(* Logix 5000 project; controller STAT 1756-L72 rev 20.12; software revision 20.04; part 15 of 34 *)
(* tags used below, declared in another part *)
   AUX_P1P2 : BOOL;
   B10 : DINT[20];
   B14 : DINT[30];
   B15 : DINT[30];
   B16 : DINT[30];
   B17 : DINT[30];
   B3 : DINT[256];
   B9 : DINT[40];
   DateTime : DINT[7];   // DINT array tag for retrieve wallclock time through GSV created during conversion
   F8 : REAL[256];
   GEN_FOUT : BOOL;
   I1_005_Bit14 : ALIAS FOR I1[5].14;
   I1_005_Bit15 : ALIAS FOR I1[5].15;
   I1_008_Bit01 : ALIAS FOR I1[8].1;   // Hand Automaat stormbekken
   I1_009_Bit04 : ALIAS FOR I1[9].4;   // Pomp 1 in lijn
   I1_009_Bit08 : ALIAS FOR I1[9].8;   // Pomp 2 in lijn
   I1_009_Bit12 : ALIAS FOR I1[9].12;   // Pomp 3 in lijn
   I1_010_Bit05 : ALIAS FOR I1[10].5;   // Vlotterschak lal stormbekken
   I2_001_Bit07 : ALIAS FOR I2[1].7;   // Motor p11 lijn1 in dienst
   I2_001_Bit09 : ALIAS FOR I2[1].9;   // Motor p12 lijn1 in dienst
   I2_001_Bit11 : ALIAS FOR I2[1].11;   // Motor p13 lijn2 in dienst
   I2_001_Bit13 : ALIAS FOR I2[1].13;   // Motor p14 lijn2 in dienst
   I2_001_Bit15 : ALIAS FOR I2[1].15;   // Motor p15 lijn3 in dienst
   I3_000_Bit00 : ALIAS FOR I3[0].0;   // Motor p15 lijn3 thermische storing
   I3_000_Bit03 : ALIAS FOR I3[0].3;   // Motor p17 lijn4 in dienst
   I3_000_Bit05 : ALIAS FOR I3[0].5;   // Motor p18 lijn4 in dienst
   I3_000_Bit09 : ALIAS FOR I3[0].9;   // Motor pro 1 voedingpomp osmose 1 in driehoek
   I3_000_Bit13 : ALIAS FOR I3[0].13;   // Motor pro 2 voedingpomp osmose 2 in driehoek
   I3_001_Bit09 : ALIAS FOR I3[1].9;   // Motor voedingspomp osmose 3 in drie
   I4_000_Bit01 : ALIAS FOR I4[0].1;   // READY DRIVE P3
   I4_000_Bit04 : ALIAS FOR I4[0].4;   // Motor p4 in lijn in
   I4_000_Bit05 : ALIAS FOR I4[0].5;   // ready drive p4
   I5_001_Bit12 : ALIAS FOR I5[1].12;   // EV6_OPEN
   I5_001_Bit13 : ALIAS FOR I5[1].13;   // EV6_TOE
   I5_001_Bit14 : ALIAS FOR I5[1].14;   // EV7_TOE
   I5_001_Bit15 : ALIAS FOR I5[1].15;   // EV7_OPEN
   I6_000_Bit13 : ALIAS FOR I6[0].13;   // ES_EV2_IS_TOE
   I6_000_Bit14 : ALIAS FOR I6[0].14;   // ES_EV2_IS_OPEN
   I7_000_Bit07 : ALIAS FOR I7[0].7;   // hoog alarm ketel tampon
   I7_000_Bit08 : ALIAS FOR I7[0].8;   // midden alarm ketel tampon
   I7_000_Bit09 : ALIAS FOR I7[0].9;   // laag alarm ketel tampon
   I7_001_Bit08 : ALIAS FOR I7[1].8;   // q4 debietsmeting osmose 1 fout
   I8_000_Bit04 : ALIAS FOR I8[0].4;   // niveau kuip 20m hoog alarm
   I8_000_Bit06 : ALIAS FOR I8[0].6;   // niveau kuip 20m laag niv
   I9_000_Bit09 : ALIAS FOR I9[0].9;   // Hand_Auto CL7
   N11 : DINT[150];
   N12 : DINT[230];
   N13 : DINT[230];
   O15_001_Bit06 : ALIAS FOR O15[1].6;   // EV2 EV2
   O15_001_Bit07 : ALIAS FOR O15[1].7;   // EV3 EV3
   O15_001_Bit10 : ALIAS FOR O15[1].10;   // EV6 EV6
   O15_001_Bit11 : ALIAS FOR O15[1].11;   // EV7 EV7
   old_o13_3 : BOOL;
   T27 : TIMER[100];
   T4 : TIMER[200];
(* ibt, continued *)

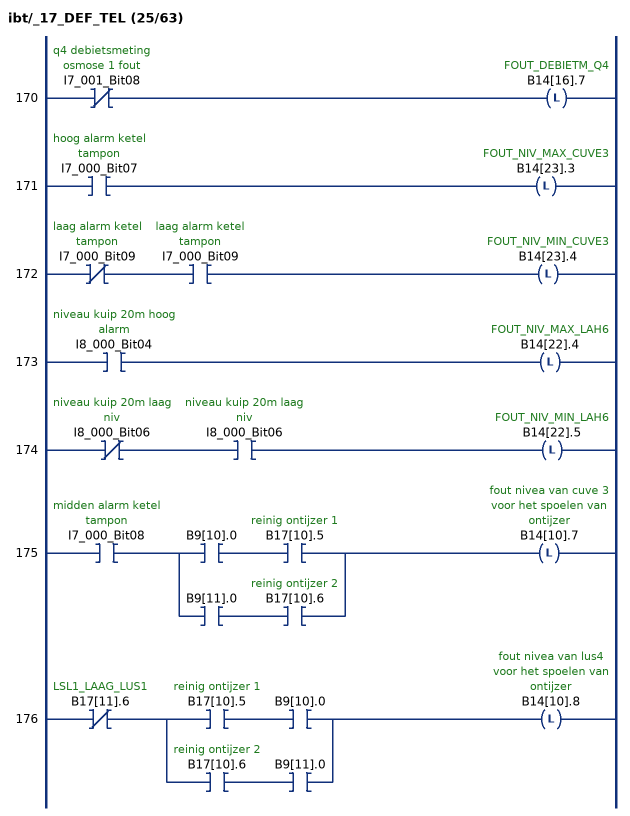
   [picture p249: ibt/_17_DEF_TEL rungs 170-176]
   170: XIO(I7_001_Bit08)OTL(B14[16].7);
   171: XIC(I7_000_Bit07)OTL(B14[23].3);
   172: XIO(I7_000_Bit09)XIC(I7_000_Bit09)OTL(B14[23].4);
   173: XIC(I8_000_Bit04)OTL(B14[22].4);
   174: XIO(I8_000_Bit06)XIC(I8_000_Bit06)OTL(B14[22].5);
   175: XIC(I7_000_Bit08)[XIC(B9[10].0) XIC(B17[10].5) ,XIC(B9[11].0) XIC(B17[10].6) ]OTL(B14[10].7);
   176: XIO(B17[11].6)[XIC(B17[10].5) XIC(B9[10].0) ,XIC(B17[10].6) XIC(B9[11].0) ]OTL(B14[10].8);
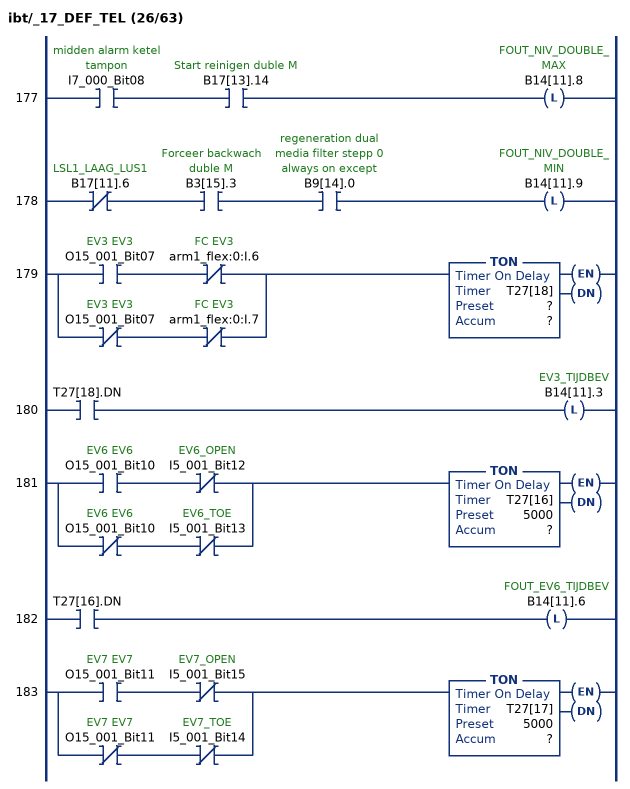
   177: XIC(I7_000_Bit08)XIC(B17[13].14)OTL(B14[11].8);
   178: XIO(B17[11].6)XIC(B3[15].3)XIC(B9[14].0)OTL(B14[11].9);
   179: [XIC(O15_001_Bit07) XIO(arm1_flex:0:I.6) ,XIO(O15_001_Bit07) XIO(arm1_flex:0:I.7) ]TON(T27[18],?,?);
   180: XIC(T27[18].DN)OTL(B14[11].3);
   181: [XIC(O15_001_Bit10) XIO(I5_001_Bit12) ,XIO(O15_001_Bit10) XIO(I5_001_Bit13) ]TON(T27[16],?,?);
   182: XIC(T27[16].DN)OTL(B14[11].6);
   183: [XIC(O15_001_Bit11) XIO(I5_001_Bit15) ,XIO(O15_001_Bit11) XIO(I5_001_Bit14) ]TON(T27[17],?,?);
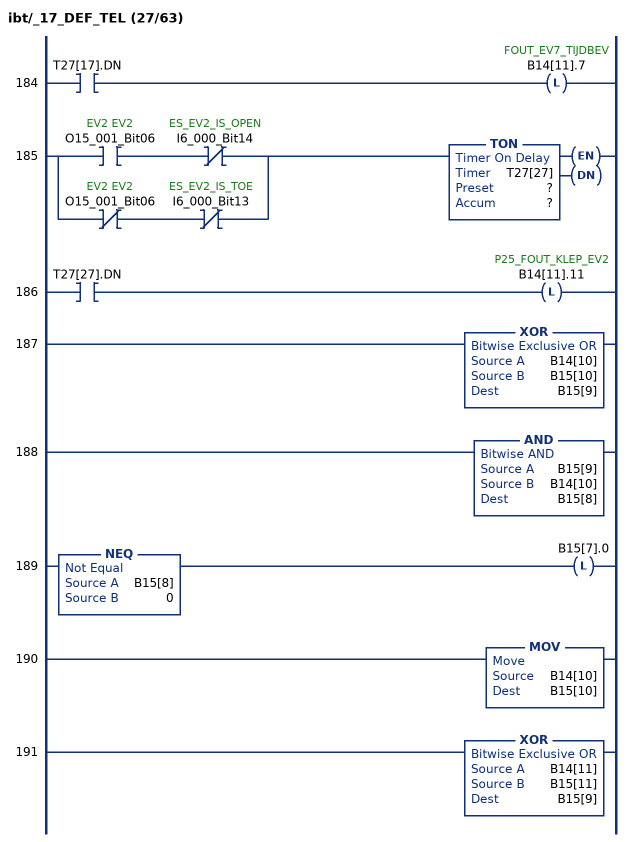
   184: XIC(T27[17].DN)OTL(B14[11].7);
   185: [XIC(O15_001_Bit06) XIO(I6_000_Bit14) ,XIO(O15_001_Bit06) XIO(I6_000_Bit13) ]TON(T27[27],?,?);
   186: XIC(T27[27].DN)OTL(B14[11].11);
   187: XOR(B14[10],B15[10],B15[9]);
   188: AND(B15[9],B14[10],B15[8]);
   189: NEQ(B15[8],0)OTL(B15[7].0);
   190: MOV(B14[10],B15[10]);
   191: XOR(B14[11],B15[11],B15[9]);
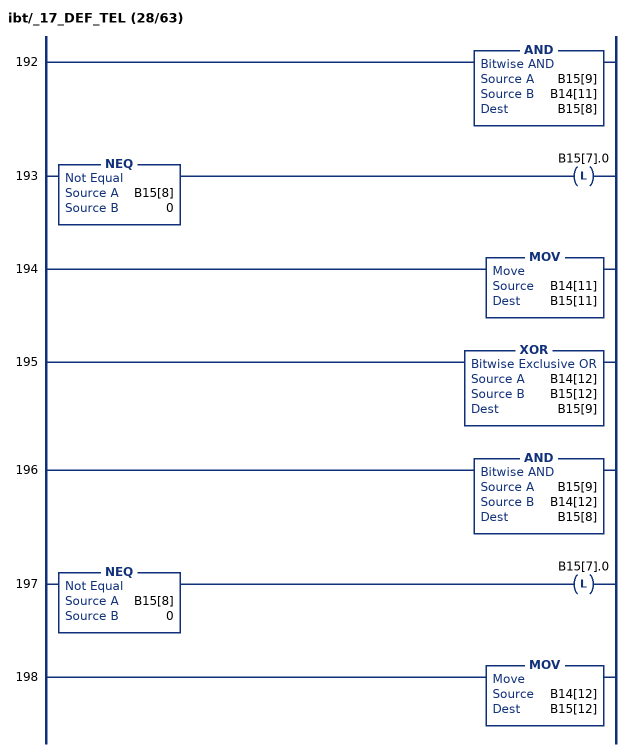
   192: AND(B15[9],B14[11],B15[8]);
   193: NEQ(B15[8],0)OTL(B15[7].0);
   194: MOV(B14[11],B15[11]);
   195: XOR(B14[12],B15[12],B15[9]);
   196: AND(B15[9],B14[12],B15[8]);
   197: NEQ(B15[8],0)OTL(B15[7].0);
   198: MOV(B14[12],B15[12]);
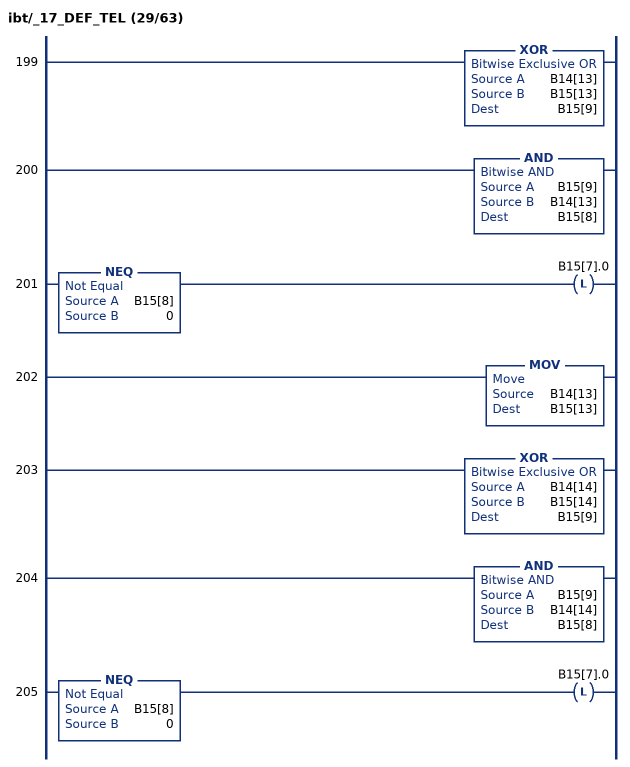
   199: XOR(B14[13],B15[13],B15[9]);
   200: AND(B15[9],B14[13],B15[8]);
   201: NEQ(B15[8],0)OTL(B15[7].0);
   202: MOV(B14[13],B15[13]);
   203: XOR(B14[14],B15[14],B15[9]);
   204: AND(B15[9],B14[14],B15[8]);
   205: NEQ(B15[8],0)OTL(B15[7].0);
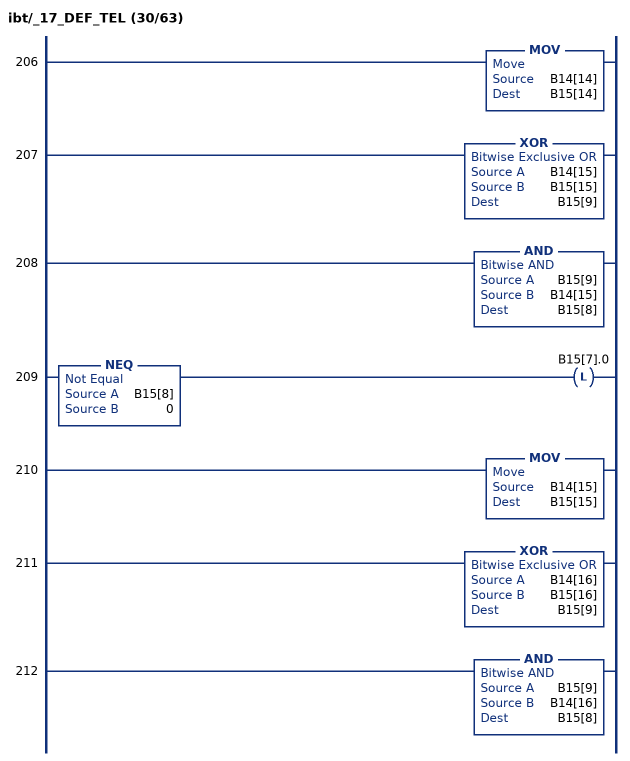
   206: MOV(B14[14],B15[14]);
   207: XOR(B14[15],B15[15],B15[9]);
   208: AND(B15[9],B14[15],B15[8]);
   209: NEQ(B15[8],0)OTL(B15[7].0);
   210: MOV(B14[15],B15[15]);
   211: XOR(B14[16],B15[16],B15[9]);
   212: AND(B15[9],B14[16],B15[8]);
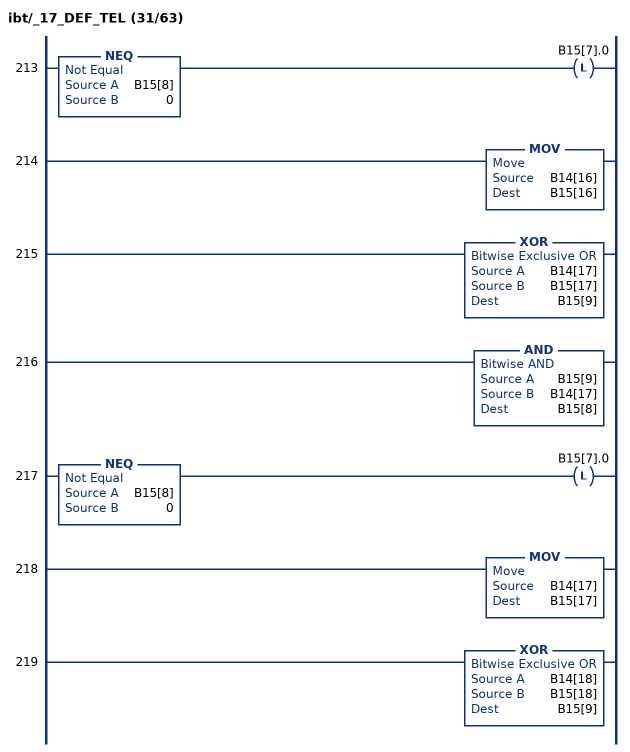
   213: NEQ(B15[8],0)OTL(B15[7].0);
   214: MOV(B14[16],B15[16]);
   215: XOR(B14[17],B15[17],B15[9]);
   216: AND(B15[9],B14[17],B15[8]);
   217: NEQ(B15[8],0)OTL(B15[7].0);
   218: MOV(B14[17],B15[17]);
   219: XOR(B14[18],B15[18],B15[9]);
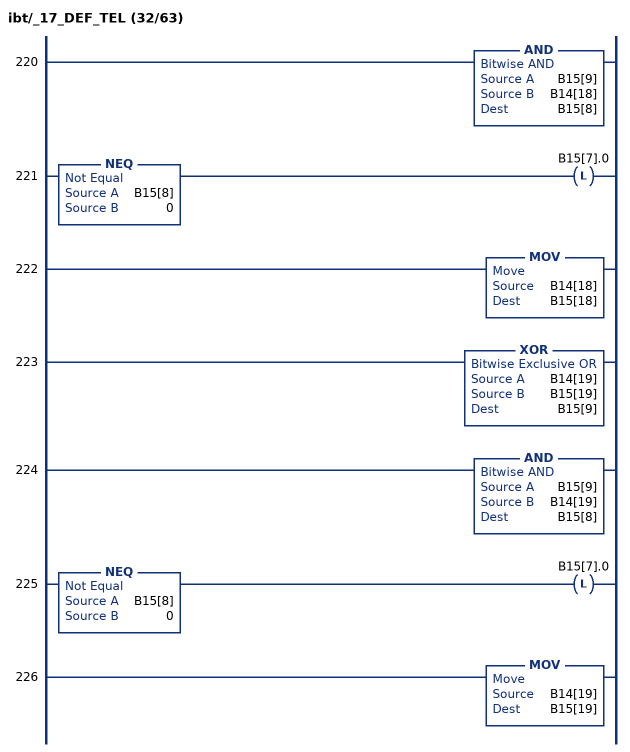
   220: AND(B15[9],B14[18],B15[8]);
   221: NEQ(B15[8],0)OTL(B15[7].0);
   222: MOV(B14[18],B15[18]);
   223: XOR(B14[19],B15[19],B15[9]);
   224: AND(B15[9],B14[19],B15[8]);
   225: NEQ(B15[8],0)OTL(B15[7].0);
   226: MOV(B14[19],B15[19]);
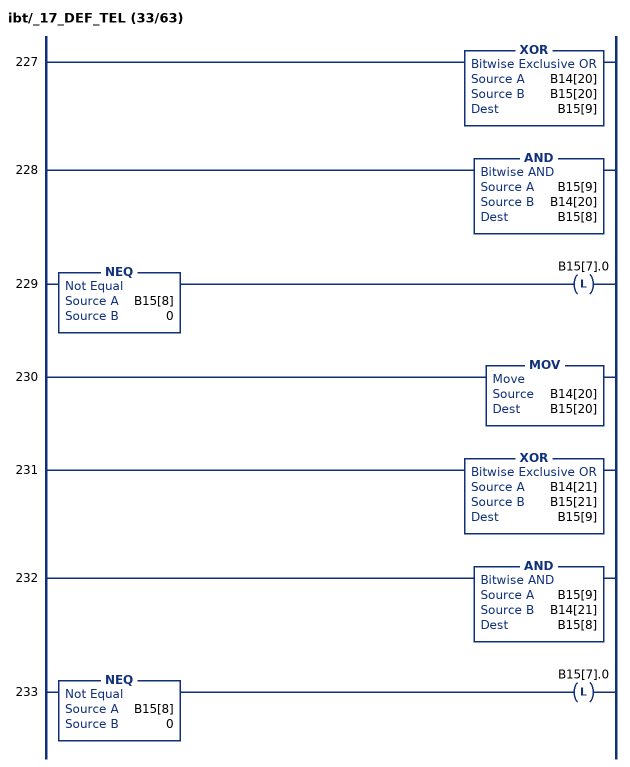
   227: XOR(B14[20],B15[20],B15[9]);
   228: AND(B15[9],B14[20],B15[8]);
   229: NEQ(B15[8],0)OTL(B15[7].0);
   230: MOV(B14[20],B15[20]);
   231: XOR(B14[21],B15[21],B15[9]);
   232: AND(B15[9],B14[21],B15[8]);
   233: NEQ(B15[8],0)OTL(B15[7].0);
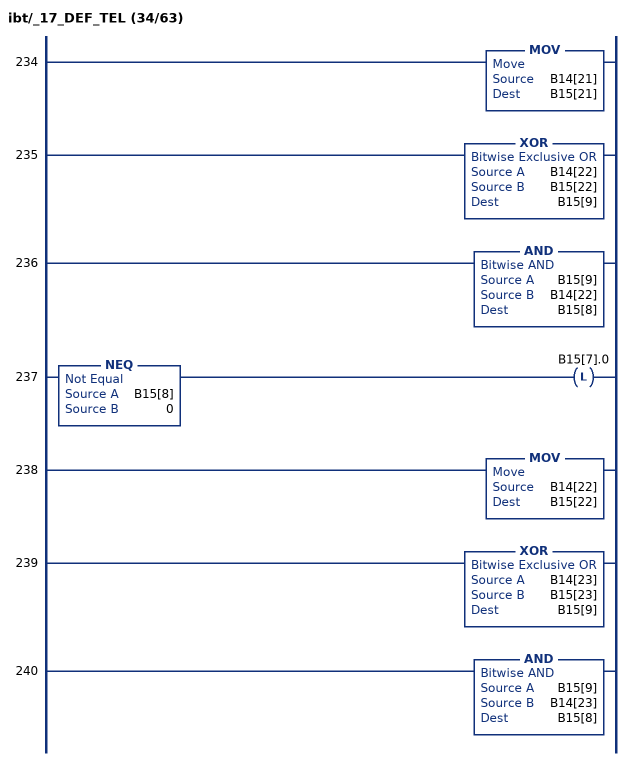
   234: MOV(B14[21],B15[21]);
   235: XOR(B14[22],B15[22],B15[9]);
   236: AND(B15[9],B14[22],B15[8]);
   237: NEQ(B15[8],0)OTL(B15[7].0);
   238: MOV(B14[22],B15[22]);
   239: XOR(B14[23],B15[23],B15[9]);
   240: AND(B15[9],B14[23],B15[8]);
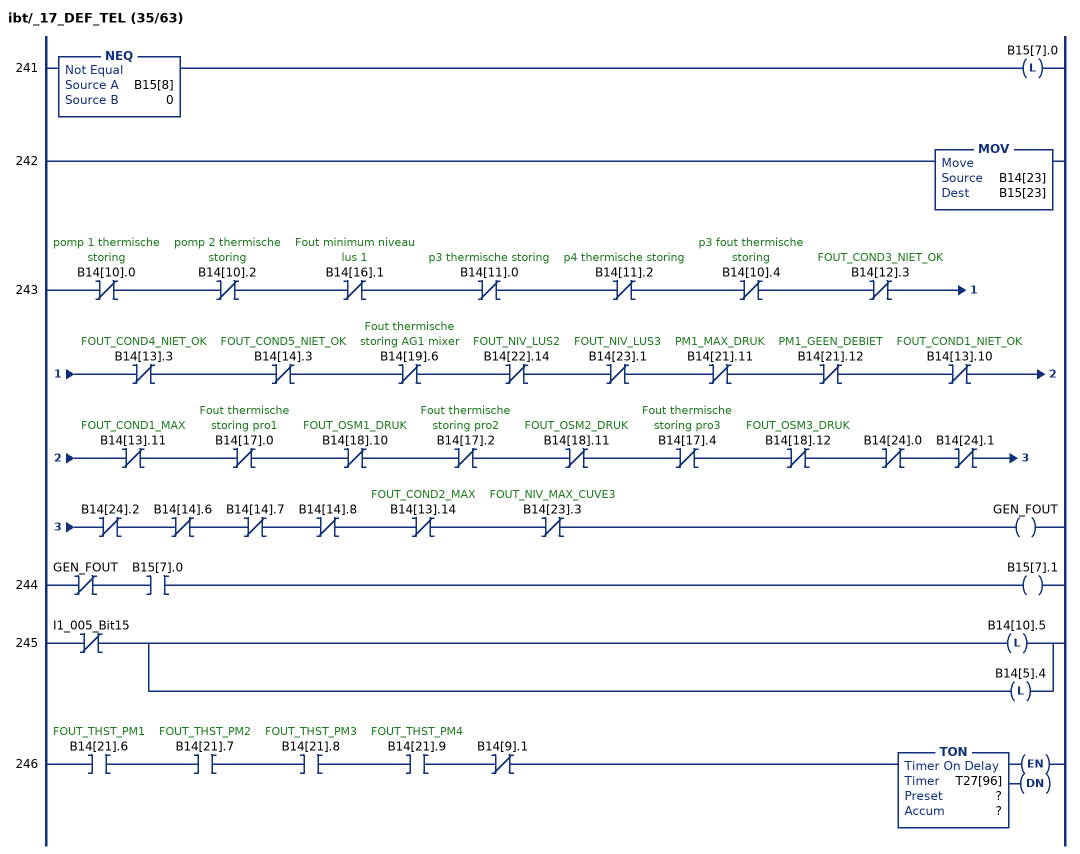
   241: NEQ(B15[8],0)OTL(B15[7].0);
   242: MOV(B14[23],B15[23]);
   243: XIO(B14[10].0)XIO(B14[10].2)XIO(B14[16].1)XIO(B14[11].0)XIO(B14[11].2)XIO(B14[10].4)XIO(B14[12].3)XIO(B14[13].3)XIO(B14[14].3)XIO(B14[19].6)XIO(B14[22].14)XIO(B14[23].1)XIO(B14[21].11)XIO(B14[21].12)XIO(B14[13].10)XIO(B14[13].11)XIO(B14[17].0)XIO(B14[18].10)XIO(B14[17].2)XIO(B14[18].11)XIO(B14[17].4)XIO(B14[18].12)XIO(B14[24].0)XIO(B14[24].1)XIO(B14[24].2)XIO(B14[14].6)XIO(B14[14].7)XIO(B14[14].8)XIO(B14[13].14)XIO(B14[23].3)OTE(GEN_FOUT);
   244: XIO(GEN_FOUT)XIC(B15[7].0)OTE(B15[7].1);
   245: XIO(I1_005_Bit15)[OTL(B14[10].5) ,OTL(B14[5].4) ];
   246: XIC(B14[21].6)XIC(B14[21].7)XIC(B14[21].8)XIC(B14[21].9)XIO(B14[9].1)TON(T27[96],?,?);
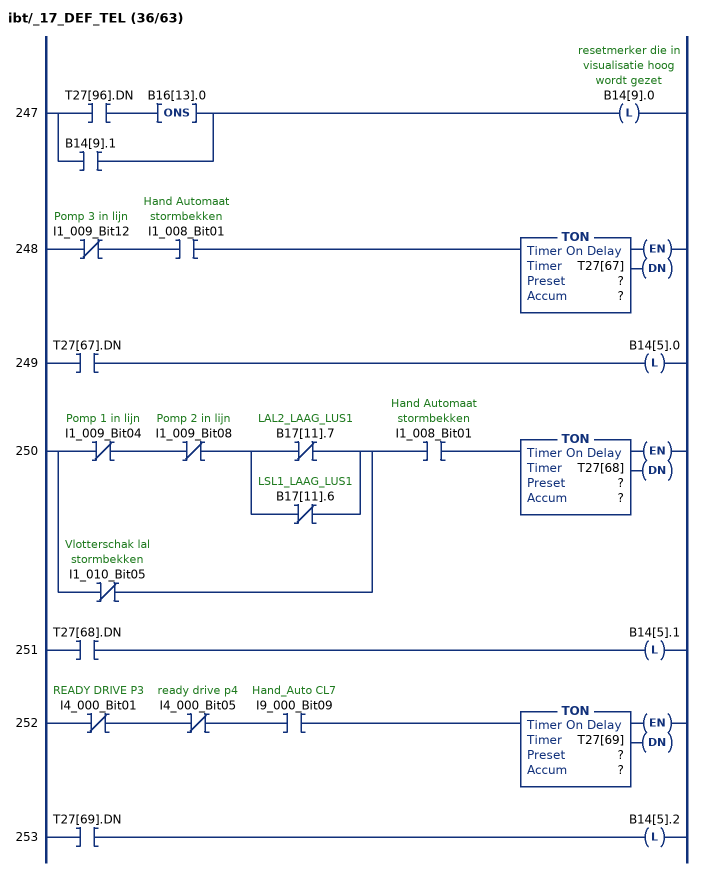
   247: [XIC(T27[96].DN) ONS(B16[13].0) ,XIC(B14[9].1) ]OTL(B14[9].0);
   248: XIO(I1_009_Bit12)XIC(I1_008_Bit01)TON(T27[67],?,?);
   249: XIC(T27[67].DN)OTL(B14[5].0);
   250: [XIO(I1_009_Bit04) XIO(I1_009_Bit08) [XIO(B17[11].7) ,XIO(B17[11].6) ] ,XIO(I1_010_Bit05) ]XIC(I1_008_Bit01)TON(T27[68],?,?);
   251: XIC(T27[68].DN)OTL(B14[5].1);
   252: XIO(I4_000_Bit01)XIO(I4_000_Bit05)XIC(I9_000_Bit09)TON(T27[69],?,?);
   253: XIC(T27[69].DN)OTL(B14[5].2);
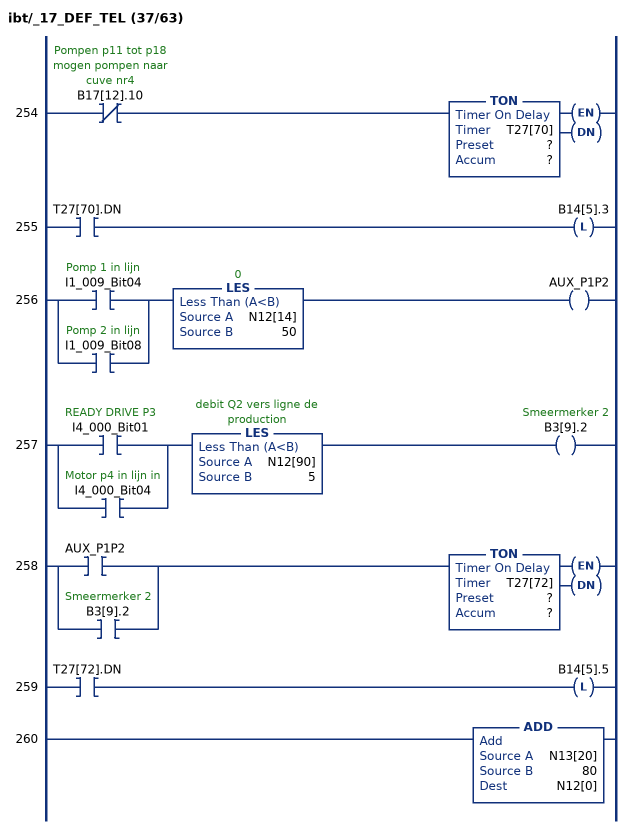
   254: XIO(B17[12].10)TON(T27[70],?,?);
   255: XIC(T27[70].DN)OTL(B14[5].3);
   256: [XIC(I1_009_Bit04) ,XIC(I1_009_Bit08) ]LES(N12[14],50)OTE(AUX_P1P2);
   257: [XIC(I4_000_Bit01) ,XIC(I4_000_Bit04) ]LES(N12[90],5)OTE(B3[9].2);
   258: [XIC(AUX_P1P2) ,XIC(B3[9].2) ]TON(T27[72],?,?);
   259: XIC(T27[72].DN)OTL(B14[5].5);
   260: ADD(N13[20],80,N12[0]);
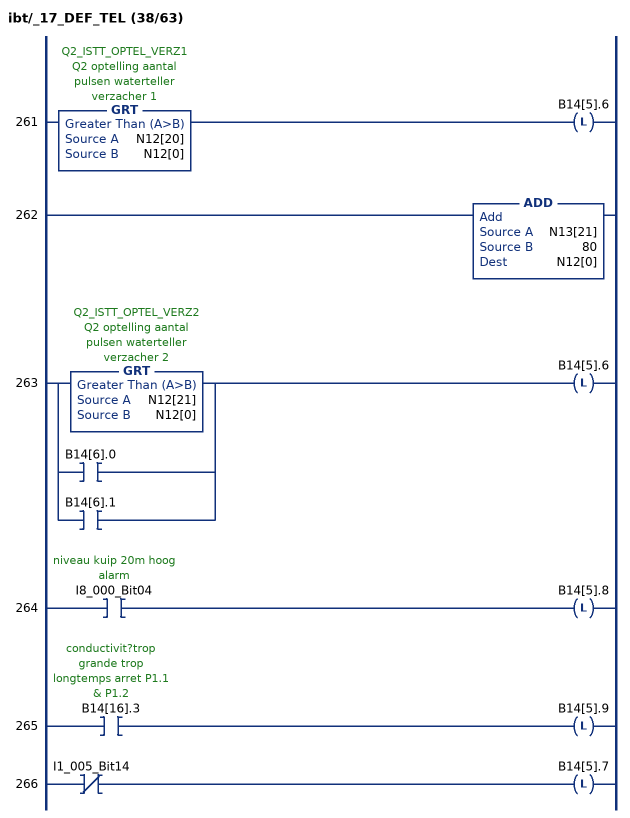
   261: GRT(N12[20],N12[0])OTL(B14[5].6);
   262: ADD(N13[21],80,N12[0]);
   263: [GRT(N12[21],N12[0]) ,[XIC(B14[6].0) ,XIC(B14[6].1) ] ]OTL(B14[5].6);
   264: XIC(I8_000_Bit04)OTL(B14[5].8);
   265: XIC(B14[16].3)OTL(B14[5].9);
   266: XIO(I1_005_Bit14)OTL(B14[5].7);
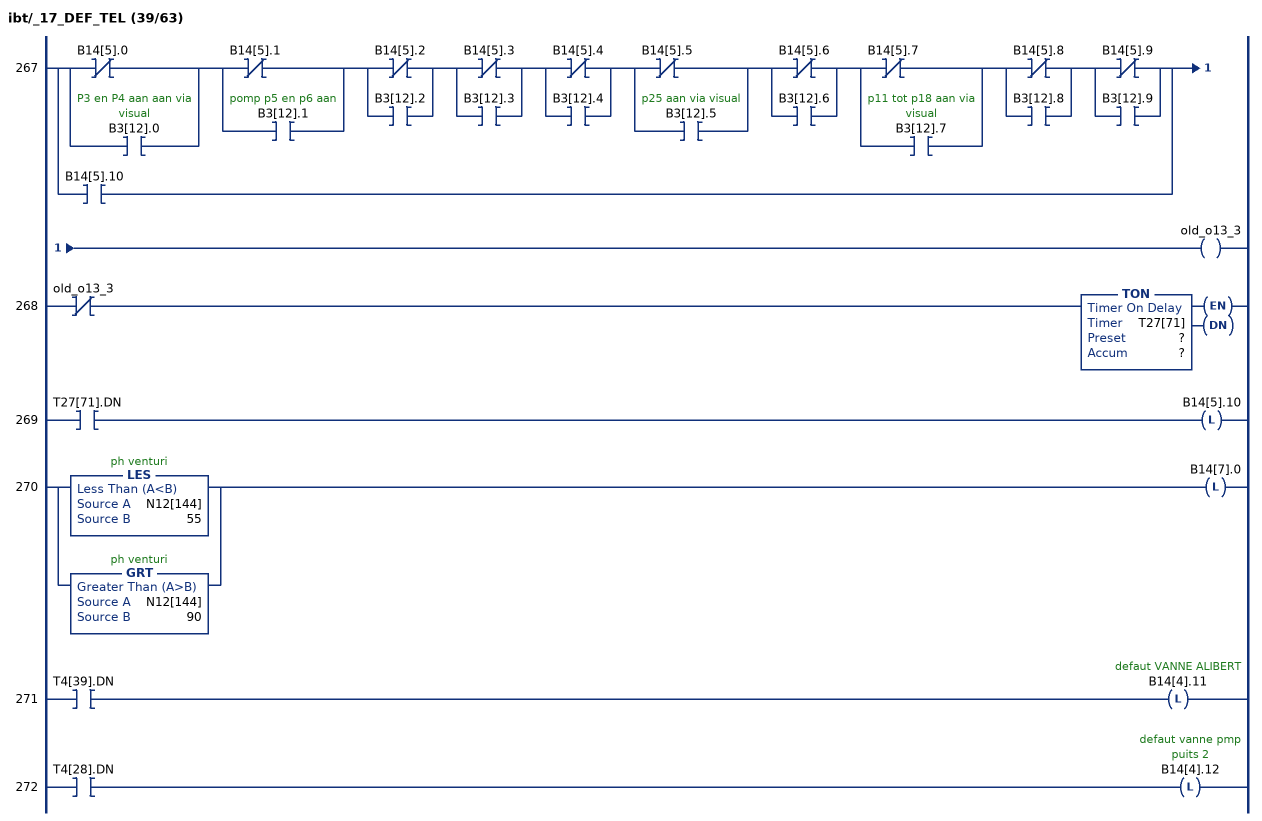
   267: [[XIO(B14[5].0) ,XIC(B3[12].0) ] [XIO(B14[5].1) ,XIC(B3[12].1) ] [XIO(B14[5].2) ,XIC(B3[12].2) ] [XIO(B14[5].3) ,XIC(B3[12].3) ] [XIO(B14[5].4) ,XIC(B3[12].4) ] [XIO(B14[5].5) ,XIC(B3[12].5) ] [XIO(B14[5].6) ,XIC(B3[12].6) ] [XIO(B14[5].7) ,XIC(B3[12].7) ] [XIO(B14[5].8) ,XIC(B3[12].8) ] [XIO(B14[5].9) ,XIC(B3[12].9) ] ,XIC(B14[5].10) ]OTE(old_o13_3);
   268: XIO(old_o13_3)TON(T27[71],?,?);
   269: XIC(T27[71].DN)OTL(B14[5].10);
   270: [LES(N12[144],55) ,GRT(N12[144],90) ]OTL(B14[7].0);
   271: XIC(T4[39].DN)OTL(B14[4].11);
   272: XIC(T4[28].DN)OTL(B14[4].12);
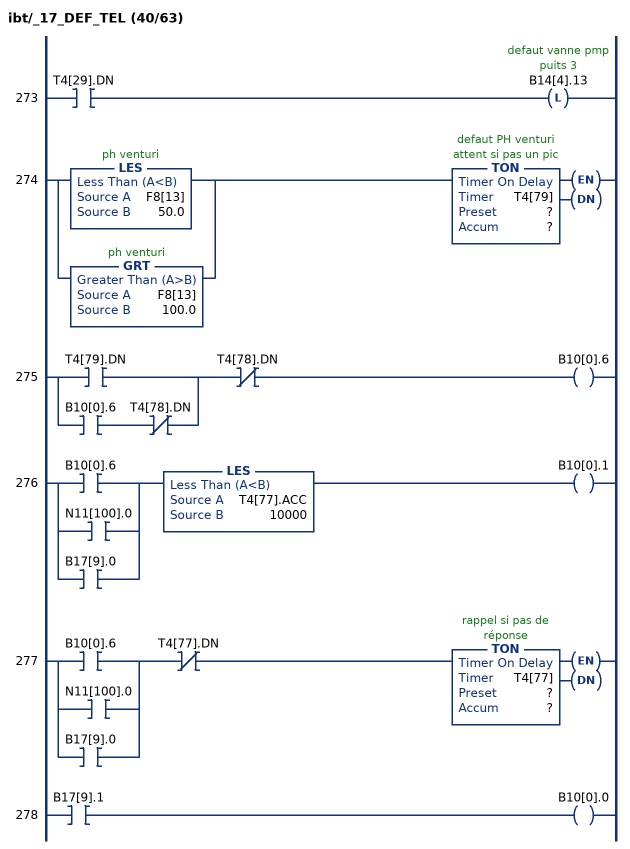
   273: XIC(T4[29].DN)OTL(B14[4].13);
   274: [LES(F8[13],50.0) ,GRT(F8[13],100.0) ]TON(T4[79],?,?);
   275: [XIC(T4[79].DN) ,XIC(B10[0].6) XIO(T4[78].DN) ]XIO(T4[78].DN)OTE(B10[0].6);
   276: [XIC(B10[0].6) ,XIC(N11[100].0) ,XIC(B17[9].0) ]LES(T4[77].ACC,10000)OTE(B10[0].1);
   277: [XIC(B10[0].6) ,XIC(N11[100].0) ,XIC(B17[9].0) ]XIO(T4[77].DN)TON(T4[77],?,?);
   278: XIC(B17[9].1)OTE(B10[0].0);
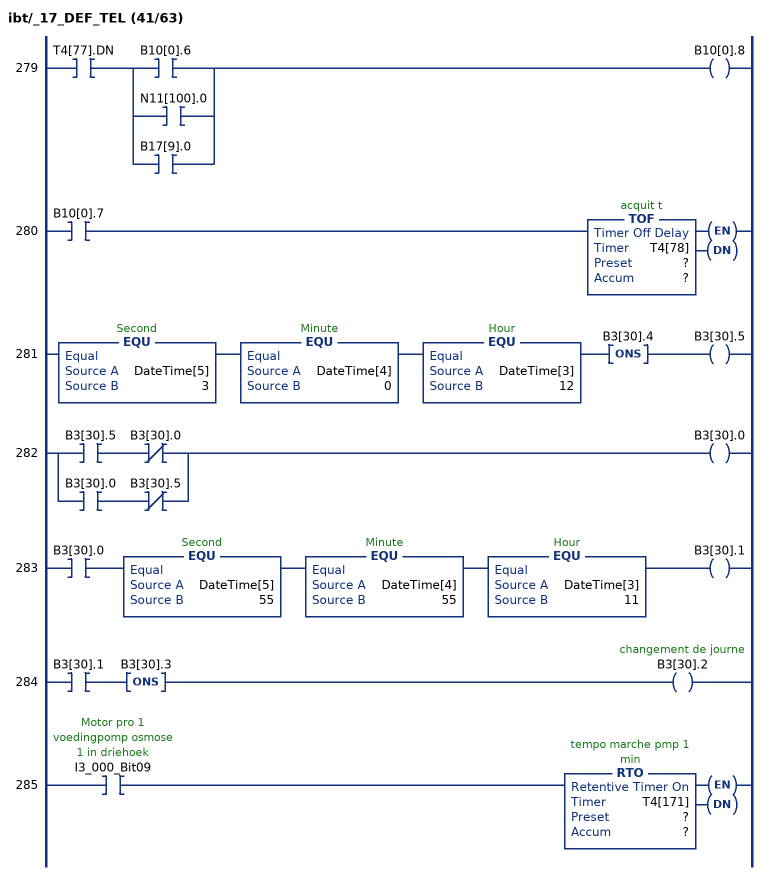
   279: XIC(T4[77].DN)[XIC(B10[0].6) ,XIC(N11[100].0) ,XIC(B17[9].0) ]OTE(B10[0].8);
   280: XIC(B10[0].7)TOF(T4[78],?,?);
   281: EQU(DateTime[5],3)EQU(DateTime[4],0)EQU(DateTime[3],12)ONS(B3[30].4)OTE(B3[30].5);
   282: [XIC(B3[30].5) XIO(B3[30].0) ,XIC(B3[30].0) XIO(B3[30].5) ]OTE(B3[30].0);
   283: XIC(B3[30].0)EQU(DateTime[5],55)EQU(DateTime[4],55)EQU(DateTime[3],11)OTE(B3[30].1);
   284: XIC(B3[30].1)ONS(B3[30].3)OTE(B3[30].2);
   285: XIC(I3_000_Bit09)RTO(T4[171],?,?);
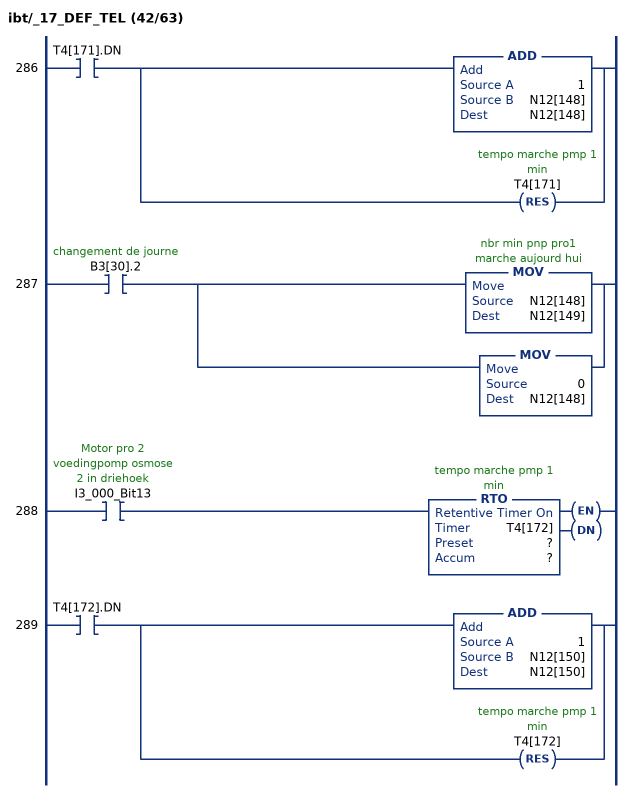
   286: XIC(T4[171].DN)[ADD(1,N12[148],N12[148]) ,RES(T4[171]) ];
   287: XIC(B3[30].2)[MOV(N12[148],N12[149]) ,MOV(0,N12[148]) ];
   288: XIC(I3_000_Bit13)RTO(T4[172],?,?);
   289: XIC(T4[172].DN)[ADD(1,N12[150],N12[150]) ,RES(T4[172]) ];
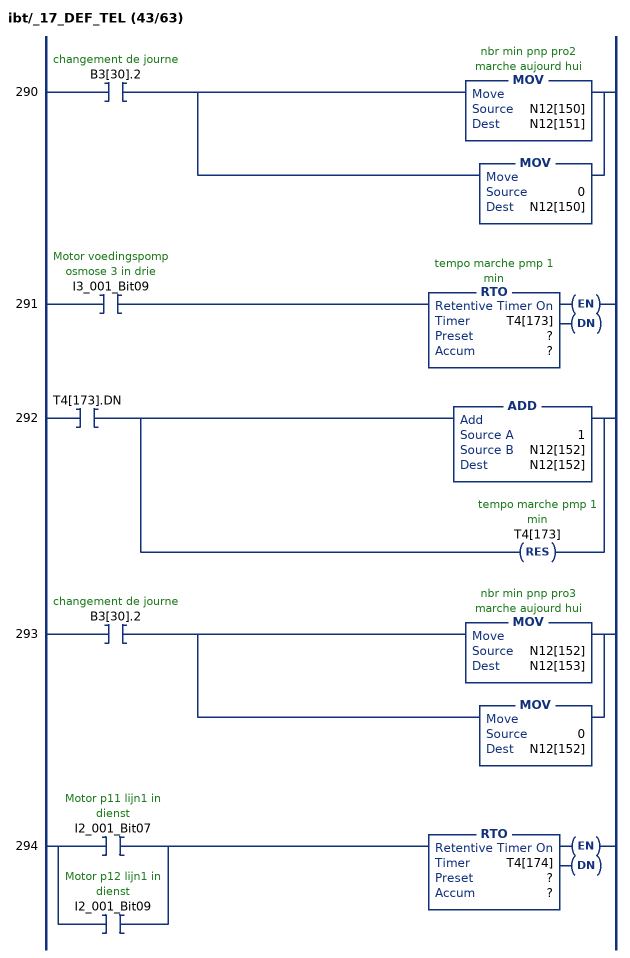
   290: XIC(B3[30].2)[MOV(N12[150],N12[151]) ,MOV(0,N12[150]) ];
   291: XIC(I3_001_Bit09)RTO(T4[173],?,?);
   292: XIC(T4[173].DN)[ADD(1,N12[152],N12[152]) ,RES(T4[173]) ];
   293: XIC(B3[30].2)[MOV(N12[152],N12[153]) ,MOV(0,N12[152]) ];
   294: [XIC(I2_001_Bit07) ,XIC(I2_001_Bit09) ]RTO(T4[174],?,?);
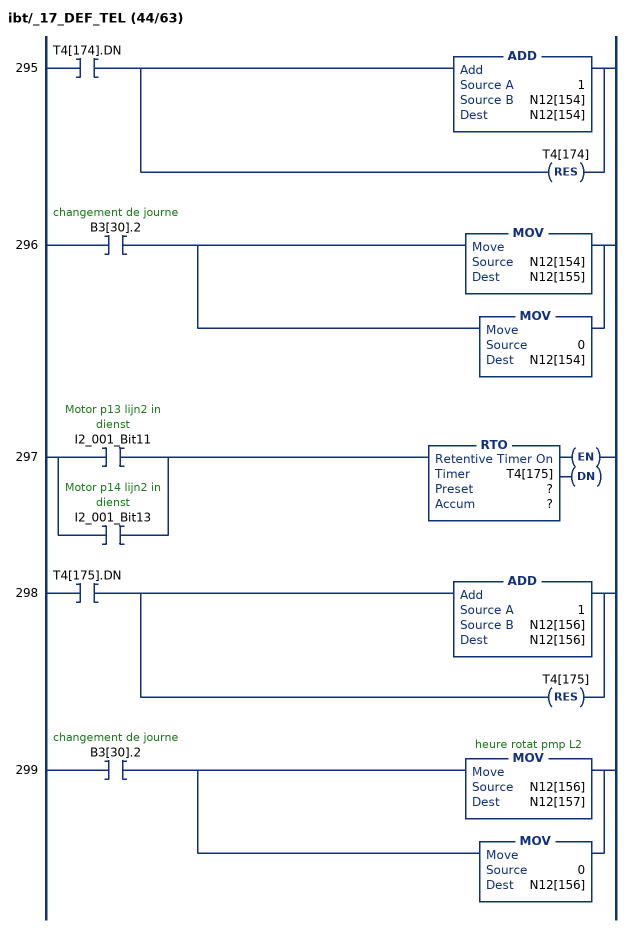
   295: XIC(T4[174].DN)[ADD(1,N12[154],N12[154]) ,RES(T4[174]) ];
   296: XIC(B3[30].2)[MOV(N12[154],N12[155]) ,MOV(0,N12[154]) ];
   297: [XIC(I2_001_Bit11) ,XIC(I2_001_Bit13) ]RTO(T4[175],?,?);
   298: XIC(T4[175].DN)[ADD(1,N12[156],N12[156]) ,RES(T4[175]) ];
   299: XIC(B3[30].2)[MOV(N12[156],N12[157]) ,MOV(0,N12[156]) ];
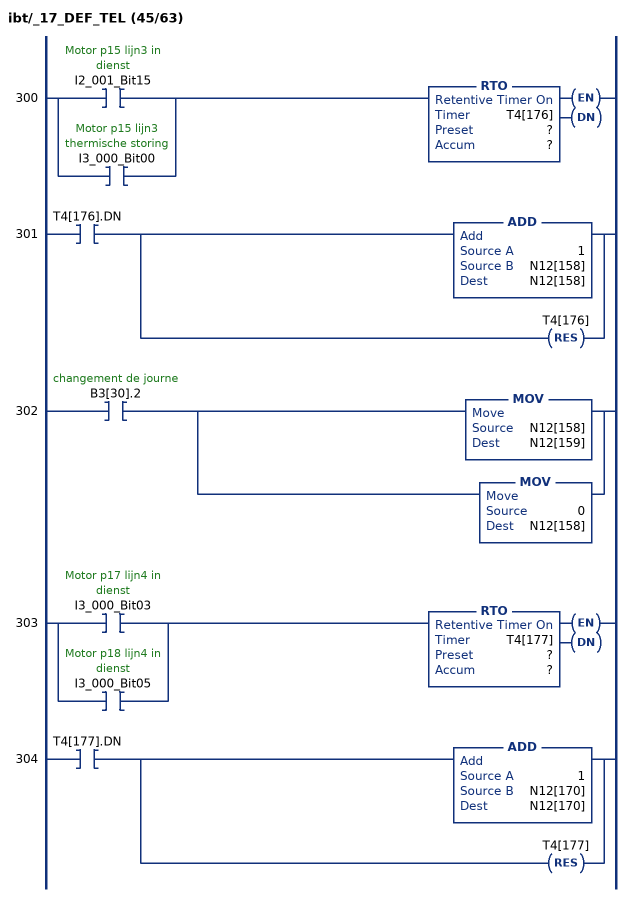
   300: [XIC(I2_001_Bit15) ,XIC(I3_000_Bit00) ]RTO(T4[176],?,?);
   301: XIC(T4[176].DN)[ADD(1,N12[158],N12[158]) ,RES(T4[176]) ];
   302: XIC(B3[30].2)[MOV(N12[158],N12[159]) ,MOV(0,N12[158]) ];
   303: [XIC(I3_000_Bit03) ,XIC(I3_000_Bit05) ]RTO(T4[177],?,?);
   304: XIC(T4[177].DN)[ADD(1,N12[170],N12[170]) ,RES(T4[177]) ];
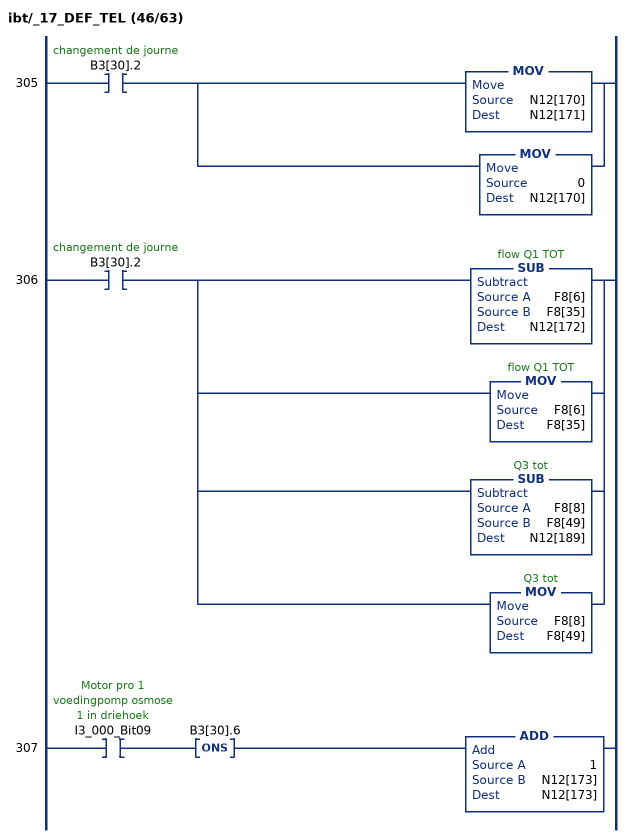
   305: XIC(B3[30].2)[MOV(N12[170],N12[171]) ,MOV(0,N12[170]) ];
   306: XIC(B3[30].2)[SUB(F8[6],F8[35],N12[172]) ,MOV(F8[6],F8[35]) ,SUB(F8[8],F8[49],N12[189]) ,MOV(F8[8],F8[49]) ];
   307: XIC(I3_000_Bit09)ONS(B3[30].6)ADD(1,N12[173],N12[173]);
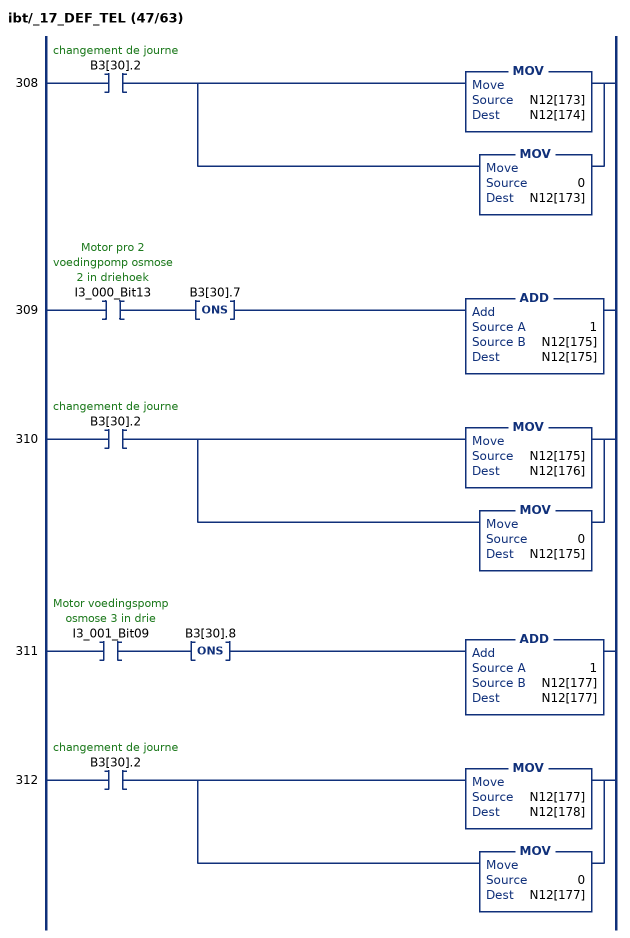
   308: XIC(B3[30].2)[MOV(N12[173],N12[174]) ,MOV(0,N12[173]) ];
   309: XIC(I3_000_Bit13)ONS(B3[30].7)ADD(1,N12[175],N12[175]);
   310: XIC(B3[30].2)[MOV(N12[175],N12[176]) ,MOV(0,N12[175]) ];
   311: XIC(I3_001_Bit09)ONS(B3[30].8)ADD(1,N12[177],N12[177]);
   312: XIC(B3[30].2)[MOV(N12[177],N12[178]) ,MOV(0,N12[177]) ];
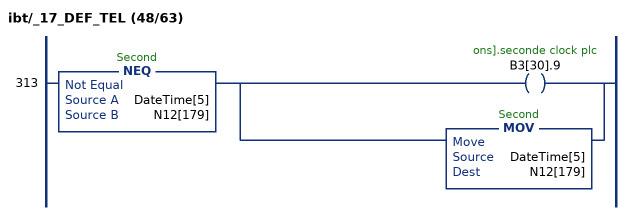
   313: NEQ(DateTime[5],N12[179])[OTE(B3[30].9) ,MOV(DateTime[5],N12[179]) ];
